// Mitsubishi GX Works2 project: PanelFlip   PLC: FX3U/FX3UC

// global labels: Global1
VAR_GLOBAL
  XXLimitN AT M8344 : BOOL;
  XXLimitP AT M8343 : BOOL;
  XXStop AT M8349 : BOOL;
  XXBusy AT M8340 : BOOL;
  XXInterruptInverse AT M8347 : BOOL;
  XXPos AT D8340 : DINT;
  XXAccelTime AT D8348 : INT;
  XXDecelTime AT D8349 : INT;
  XXLimitNView AT M0 : BOOL;
  XXLimitPView AT M1 : BOOL;
  XXPosView AT D0 : DINT;
  XXTarPos AT D2 : DINT;
  XXFeed AT D4 : DINT;
  XXTarR AT M2 : BOOL;
  XXTarRSkip AT D6 : INT;
  XXManualN AT M3 : BOOL;
  XXManualP AT M4 : BOOL;
  XXOn AT M5 : BOOL;
  XXRun AT M6 : BOOL;
  XXDirection AT M7 : BOOL;
  XXMinI AT X000 : BOOL;
  XXAlarmI AT X004 : BOOL;
  XXReadyI AT X010 : BOOL;
  XXLimitNI AT X011 : BOOL;
  XXLimitPI AT X012 : BOOL;
  XXPulseO AT Y000 : BOOL;
  XXDirectionO AT Y004 : BOOL;
  XXOnO AT Y002 : BOOL;
  MachineReady AT M8 : BOOL;
  MachineReadyTimer AT TC0 : BOOL;
  DataState AT D7 : INT;
  Run AT M9 : BOOL;
  RunStop AT M10 : BOOL;
  RunReset AT M11 : BOOL;
  RunState AT D8 : INT;
  RunStateNext AT M12 : BOOL;
  RunStateBase AT D9 : INT;
  RunStateBaseNext AT M13 : BOOL;
  RunStateGrab AT D10 : INT;
  RunStateGrabNext AT M14 : BOOL;
  RunStateFlip AT D11 : INT;
  RunStateFlipNext AT M15 : BOOL;
  FlipFoilIn AT M16 : BOOL;
  FlipFoilInI AT X001 : BOOL;
  FlipFoilInIPulseCatch AT M8171 : BOOL;
  FlipFoilInIDenoiseTimer AT TC1 : BOOL;
  FlipEnd AT M17 : BOOL;
  FlipEndI AT X002 : BOOL;
  FlipEndIPulseCatch AT M8172 : BOOL;
  RS485Index AT D12 : INT;
  RS485Timer AT TC2 : BOOL;
  RS485RW : RS485RW;
  RS485Send0 AT D13 : INT;
  RS485Send1 AT D14 : INT;
  RS485Send2 AT D15 : INT;
  RS485Send3 AT D16 : INT;
  RS485Send4 AT D17 : INT;
  RS485Send5 AT D18 : INT;
  RS485Send6 AT D19 : INT;
  RS485Send7 AT D20 : INT;
  RS485Send8 AT D21 : INT;
  RS485Send9 AT D22 : INT;
  RS485Send10 AT D23 : INT;
  RS485Send11 AT D24 : INT;
  RS485Send12 AT D25 : INT;
  RS485Send13 AT D26 : INT;
  RS485Send14 AT D27 : INT;
  RS485Send15 AT D28 : INT;
  RS485Send16 AT D29 : INT;
  RS485Send17 AT D30 : INT;
  RS485Send18 AT D31 : INT;
  RS485Send19 AT D32 : INT;
  RS485Receive0 AT D33 : INT;
  RS485Receive1 AT D34 : INT;
  RS485Receive2 AT D35 : INT;
  RS485Receive3 AT D36 : INT;
  RS485Receive4 AT D37 : INT;
  RS485Receive5 AT D38 : INT;
  RS485Receive6 AT D39 : INT;
  RS485Receive7 AT D40 : INT;
  RS485Receive8 AT D41 : INT;
  RS485Receive9 AT D42 : INT;
  RS485Receive10 AT D43 : INT;
  RS485Receive11 AT D44 : INT;
  RS485Receive12 AT D45 : INT;
  RS485Receive13 AT D46 : INT;
  RS485Receive14 AT D47 : INT;
  RS485Receive15 AT D48 : INT;
  RS485Receive16 AT D49 : INT;
  RS485Receive17 AT D50 : INT;
  RS485Receive18 AT D51 : INT;
  RS485Receive19 AT D52 : INT;
  SpindleFlipRun AT M18 : BOOL;
  SpindleFlipRunO AT Y014 : BOOL;
  SpindleBeltRun AT M19 : BOOL;
  SpindleBeltRunO AT Y015 : BOOL;
  SpindleFlip_W_HzValue0 AT D53 : INT;
  SpindleBelt_W_HzValue1 AT D54 : INT;
  SpindleFlip_W_RunValue2 AT D55 : INT;
  SpindleBelt_W_RunValue3 AT D56 : INT;
  SpindleFlip_R_HzValue4 AT D57 : INT;
  SpindleBelt_R_HzValue5 AT D58 : INT;
  SpindleFlip_R_SetHzValue6 AT D59 : INT;
  SpindleBelt_R_SetHzValue7 AT D60 : INT;
  SpindleFlip_R_BusVValue8 AT D61 : INT;
  SpindleBelt_R_BusVValue9 AT D62 : INT;
  SpindleFlip_R_OutVValue10 AT D63 : INT;
  SpindleBelt_R_OutVValue11 AT D64 : INT;
  SpindleFlip_R_OutCValue12 AT D65 : INT;
  SpindleBelt_R_OutCValue13 AT D66 : INT;
  RS485SpindleFlip_W_Hz0 AT M20 : BOOL;
  RS485SpindleBelt_W_Hz1 AT M21 : BOOL;
  RS485SpindleFlip_W_Run2 AT M22 : BOOL;
  RS485SpindleBelt_W_Run3 AT M23 : BOOL;
  RS485SpindleFlip_R_Hz4 AT M24 : BOOL;
  RS485SpindleBelt_R_Hz5 AT M25 : BOOL;
  RS485SpindleFlip_R_SetHz6 AT M26 : BOOL;
  RS485SpindleBelt_R_SetHz7 AT M27 : BOOL;
  RS485SpindleFlip_R_BusV8 AT M28 : BOOL;
  RS485SpindleBelt_R_BusV9 AT M29 : BOOL;
  RS485SpindleFlip_R_OutV10 AT M30 : BOOL;
  RS485SpindleBelt_R_OutV11 AT M31 : BOOL;
  RS485SpindleFlip_R_OutC12 AT M32 : BOOL;
  RS485SpindleBelt_R_OutC13 AT M33 : BOOL;
  RS485Dummy14 AT M34 : BOOL;
  RS485Dummy15 AT M35 : BOOL;
  GrabMoveStart AT D67 : DINT;
  GrabMoveEnd AT D69 : DINT;
  GrabMoveSpeed AT D71 : DINT;
  GrabMoveAccelTime AT D73 : INT;
  GrabMoveDecelTime AT D74 : INT;
  GrabDownMin AT M36 : BOOL;
  GrabDownMinI AT X005 : BOOL;
  GrabDownMax AT M37 : BOOL;
  GrabDownMaxI AT X006 : BOOL;
  GrabDown AT M38 : BOOL;
  GrabDownO AT Y005 : BOOL;
  GrabDownATimer AT TC3 : BOOL;
  GrabDownATimerDelay AT D75 : INT;
  GrabDownBTimer AT TC4 : BOOL;
  GrabDownBTimerDelay AT D76 : INT;
  GrabDownCTimer AT TC5 : BOOL;
  GrabDownCTimerDelay AT D77 : INT;
  GrabDownDTimer AT TC6 : BOOL;
  GrabDownDTimerDelay AT D78 : INT;
  GrabDownCXTimer AT TC7 : BOOL;
  GrabOn1 AT M39 : BOOL;
  GrabOn2 AT M40 : BOOL;
  GrabOn3 AT M41 : BOOL;
  GrabOn4 AT M42 : BOOL;
  GrabOn5 AT M43 : BOOL;
  GrabOn1O AT Y006 : BOOL;
  GrabOn2O AT Y010 : BOOL;
  GrabOn3O AT Y011 : BOOL;
  GrabOn4O AT Y012 : BOOL;
  GrabOn5O AT Y013 : BOOL;
  GrabOnTimer AT TC8 : BOOL;
  GrabOnTimerDelay AT D79 : INT;
  GrabOnIndex AT D80 : INT;
  GrabPump AT M44 : BOOL;
  GrabPumpO AT Y007 : BOOL;
  GrabManualEnable AT M45 : BOOL;
  GrabStepReady AT M46 : BOOL;
  BaseEmpty AT M47 : BOOL;
  BaseEmptyI AT X003 : BOOL;
  MirrorI AT X007 : BOOL;
  M8012PLS AT M48 : BOOL;
  TestGrabDownEnable AT M49 : BOOL;
  TestGrabDownMinTimer AT TC9 : BOOL;
  TestGrabDownMaxTimer AT TC10 : BOOL;
END_VAR

// task Task_01 (event TRUE, interval 0, priority 31): POU_01

PROGRAM POU_01
VAR
  fTmp : BOOL;
END_VAR
SET(M8002, M8336);
MOV(M8002, HFFF0, D8336);
SET(M8002, XXInterruptInverse);
ZRST(M8002, RunState, RunStateFlip);
MOV(M8002, 200, XXAccelTime);
MOV(M8002, 200, XXDecelTime);
RST(M8002, SpindleFlipRun);
RST(M8002, SpindleBeltRun);
RST(M8002, TestGrabDownEnable);

(*ready*)
RST(M8002, MachineReady);
OUT_T(NOT MachineReady, MachineReadyTimer, 10);
SET(MachineReadyTimer, MachineReady);

(*data*)
RST(M8002, DataState);
DECO(M8000, DataState, 3, M500); (*M500 - M507*)
MOV(M501, GrabMoveAccelTime, XXAccelTime);
MOV(M501, GrabMoveDecelTime, XXDecelTime);
MOV(M501, 2, DataState); (*jump to rs485 sync data*)

SET(M507 AND RunState = 0 AND Run , fTmp);
RST(fTmp, Run);
RST(fTmp, RunStop);
MOV(fTmp, 1, RunState);
RST(fTmp, fTmp);
SET(RunState > 0 AND RunReset, fTmp);
RST(fTmp, RunReset);
RST(fTmP, RunStop);
RST(fTmp, Run);
RST(fTmp, SpindleFlipRun);
RST(fTmp, SpindleBeltRun);
RST(fTmp, XXRun);
ZRST(fTmp, GrabOn1, GrabOn5);
ZRST(fTmp, RunState, RunStateFlip);
ZRST(fTmp, RunStateNext, RunStateFlipNext);
RST(fTmp, fTmp);

INC(RunStateNext, RunState);
INC(RunStateBaseNext, RunStateBase);
INC(RunStateGrabNext, RunStateGrab);
INC(RunStateFlipNext, RunStateFlip);
ZRST(M8000, RunStateNext, RunStateFlipNext);
DECO(M8000, RunState, 6, M100); 
DECO(M8000, RunStateBase, 6, M200);
DECO(M8000, RunStateGrab, 6, M300); DECO(M8000, RunStateGrab, 6, M1300); ZRST(NOT (XXTarR AND XXReadyI), M1300, M1363);
DECO(M8000, RunStateFlip, 6, M400);

(*||||||||||*)
(*||||||||||Main*)
(*start belt*)
SET(M101, SpindleBeltRun);
SET(M101, RunStateNext);
(*start belt done, start other*)
MOV(M102 AND M200, 1, RunStateBase);
MOV(M102 AND M1300, 1, RunStateGrab);
MOV(M102 AND M400, 1, RunStateFlip);
MOV(M102, 10, RunState);
(*run or stop, auto or manual*)
SET(M110 AND RunStop AND NOT BaseEmpty AND Run, fTmp);
RST(fTmp, RunStop);
RST(fTmp, Run);
RST(fTmp, fTmp);
SET(M110 AND NOT RunStop, fTmp);
MOV(fTmp AND NOT GrabManualEnable, 11, RunState);
MOV(fTmp AND GrabManualEnable, 21, RunState);
DECOP(fTmp, RunState, 6, M100);
RST(fTmp, fTmp);
(*auto*)
SET(M111 AND M1340, fTmp);
MOV(fTmp AND NOT RunStop, 11, RunStateGrab);
MOV(fTmp, 10, RunState);
SET(fTmp, GrabStepReady);
RST(fTmp, fTmp);
(*manual*)
SET(M121 AND M1340, fTmp);
MOV(fTmp AND NOT RunStop, 11, RunStateGrab);
MOV(fTmp, 10, RunState);
RST(fTmp, fTmp);
(*/////base and flip*)
(*seperate sequence*)
MOV(M219 OR M220, 11, RunStateBase);
MOV(M420, 11, RunStateFlip);

(*||||||||||*)
(*||||||||||Base*)
(*/////reset*)
MOV(M201, 11, RunStateBase);
(*empty, stop*)
MOV(M211 AND BaseEmpty, 19, RunStateBase);
SET(M211 AND BaseEmpty, RunStop);
(*not empty, ready*)
MOV(M211 AND NOT BaseEmpty, 20, RunStateBase);
(*||||||||||*)

(*||||||||||*)
(*||||||||||Grab*)
(*/////reset*)
(*1 pulse = 0.01 mm*)
(*turn servo on, grab up off all*)
SET(M301 AND NOT XXOn, XXOn);
RST(M301, GrabDown);
ZRST(M301, GrabOn1, GrabOn5);
SET(M1301 AND GrabDownMin, RunStateGrabNext);
(*min on, jump to dvit*)
MOV(M1302 AND XXMinI, 5, RunStateGrab);
(*min off, jump to move back*)
SET(M1302 AND NOT XXMinI, RunStateGrabNext);
(*move back*)
RST(M1303, XXPos);
DMOV(M1303, -3000_00, XXTarPos);
DMOV(M1303, 100_00, XXFeed);
SET(M1303, XXRun);
SET(M1303, RunStateGrabNext);
(*move back hit min, jump to dvit*)
RST(M304 AND XXMinI, XXRun);
MOV(M1304 AND XXMinI, 5, RunStateGrab);
(*dvit*)
DDVIT(M305, 10_00, 10_00, XXPulseO, XXDirection);
SET(M305 AND M8029, RunStateGrabNext);
RST(M305 AND M8029, M305);
(*get origin done, jump to (move to start position)*)
RST(M1306, XXPos);
RST(M1306, XXTarPos);
MOV(M1306, 30, RunStateGrab);
(*/////work sequence*)
(*move to start position*)
DMOV(M1311, GrabMoveStart, XXTarPos);
DMOV(M1311, GrabMoveSpeed, XXFeed);
SET(M1311, XXRun);
SET(M1311, RunStateGrabNext);
(*grab down on all, reset grab on index*)
SET(M1312, GrabDown);
SET(M1312, GrabOn1);
SET(M1312, GrabOn2);
SET(M1312, GrabOn3);
SET(M1312, GrabOn4);
SET(M1312, GrabOn5);
RST(M1312, GrabOnIndex);
SET(M1312 AND GrabDownMax, RunStateGrabNext);
(*wait A*)
OUT_T(M1313, GrabDownATimer, GrabDownATimerDelay);
SET(GrabDownATimer, RunStateGrabNext);
(*grab up*)
RST(M1314, GrabDown);
SET(M1314 AND GrabDownMin, RunStateGrabNext);
(*wait B*)
OUT_T(M1315, GrabDownBTimer, GrabDownBTimerDelay);
SET(GrabDownBTimer, RunStateGrabNext);
(*move to end position*)
DMOV(M1316, GrabMoveEnd, XXTarPos);
DMOV(M1316, GrabMoveSpeed, XXFeed);
SET(M1316, XXRun);
SET(M1316, RunStateGrabNext);
(*wait C*)
OUT_T(M1317, GrabDownCTimer, GrabDownCTimerDelay);
SET(GrabDownCTimer, RunStateGrabNext);
(*grab down*)
SET(M1318, GrabDown);
SET(M1318 AND GrabDownMax, RunStateGrabNext);
(*wait D*)
OUT_T(M1319, GrabDownDTimer, GrabDownDTimerDelay);
SET(GrabDownDTimer, RunStateGrabNext);
(*drop start*)
SET(M1320, RunStateGrabNext);
(*drop and check*)
OUT_T(M1321, GrabOnTimer, GrabOnTimerDelay);
SET(M1321 AND (GrabOnTimer OR GrabOnIndex = 0), fTmp);
RST(fTmp AND NOT MirrorI AND GrabOnIndex = 0, GrabOn1);
RST(fTmp AND NOT MirrorI AND GrabOnIndex = 1, GrabOn2);
RST(fTmp AND NOT MirrorI AND GrabOnIndex = 2, GrabOn3);
RST(fTmp AND NOT MirrorI AND GrabOnIndex = 3, GrabOn4);
RST(fTmp AND NOT MirrorI AND GrabOnIndex = 4, GrabOn5);
RST(fTmp AND MirrorI AND GrabOnIndex = 0, GrabOn5);
RST(fTmp AND MirrorI AND GrabOnIndex = 1, GrabOn4);
RST(fTmp AND MirrorI AND GrabOnIndex = 2, GrabOn3);
RST(fTmp AND MirrorI AND GrabOnIndex = 3, GrabOn2);
RST(fTmp AND MirrorI AND GrabOnIndex = 4, GrabOn1);
INC(fTmp, GrabOnIndex);
MOV(fTmp AND GrabOnIndex < 5, 20, RunStateGrab); (*jump back to (drop start)*)
MOV(fTmp AND GrabOnIndex >= 5, 22, RunStateGrab); (*drop done, use move because manual ignore RunStateGrabNext*)
RST(fTmp, fTmp);
(*grab up*)
RST(M1322, GrabDown);
SET(M1322 AND GrabDownMin, RunStateGrabNext);
(*wait C*)
OUT_T(M1323, GrabDownCXTimer, GrabDownCTimerDelay);
MOV(GrabDownCXTimer, 30, RunStateGrab);
(*move to start position*)
DMOV(M1330, GrabMoveStart, XXTarPos);
DMOV(M1330, GrabMoveSpeed, XXFeed);
SET(M1330, XXRun);
SET(M1330, RunStateGrabNext);
(*move to start position done, end*)
MOV(M1331, 40, RunStateGrab);
(*/////*)
(*manual*)
SET(GrabManualEnable AND RunStateGrabNext AND RunStateGrab > 10, fTmp);
RST(fTmp AND NOT GrabStepReady, RunStateGrabNext);
RST(fTmp AND GrabStepReady, GrabStepReady);
RST(fTmp, fTmp);
(*||||||||||*)

(*||||||||||*)
(*||||||||||Flip*)
(*/////reset*)
(*rotate, forward = 1, reverse = 2, stop = 5*)
SET(M401, SpindleFlipRun);
RST(M401, FlipEndIPulseCatch);
SET(M401, RunStateFlipNext);
(*stop rotate*)
SET(M402 AND FlipEnd, fTmp);
RST(fTmp, SpindleFlipRun);
RST(fTmp, FlipFoilInIPulseCatch);
RST(fTmp, FlipEndIPulseCatch);
MOV(fTmp, 11, RunStateFlip);
RST(fTmp, fTmp);
(*/////work sequence*)
(*foil in, rotate*)
SET(M411 AND FlipFoilIn, fTmp);
SET(fTmp, SpindleFlipRun);
RST(fTmp, FlipFoilInIPulseCatch);
RST(fTmp, FlipFoilIn);
RST(fTmp, FlipEndIPulseCatch);
SET(fTmp, RunStateFlipNext);
RST(fTmp, fTmp);
(*stop rotate*)
SET(M412 AND FlipEnd, fTmp);
RST(fTmp, SpindleFlipRun);
RST(fTmp, FlipFoilInIPulseCatch);
RST(fTmp, FlipFoilIn);
RST(fTmp, FlipEndIPulseCatch);
MOV(fTmp, 20, RunStateFlip);
RST(fTmp, fTmp);
(*||||||||||*)

(*||||||||||*)
(*||||||||||RS485*)
(*combine 2 register first 8bit data to 16bit register example: MOV(D0(High), K2M8), MOV(D1(Low), K2M0) then MOV(K4M0, D2) now D2 is combination of D0 and D1*)
(*main*)
MOV(M8002, H0C87, D8120);
MOV(M8002, K1000, D8129);
SET(M8002, M8161);
RS(M8012, RS485Send0, K8, K11, RS485Receive0);
PLS(M8012, M8012PLS); SET(M8012PLS, M8122);
RST(M8123, M8123);
(*sync data*)
DECO(M8000, RS485Index, 4, RS485SpindleFlip_W_Hz0);
(*start, set first index*)
MOV(M502, 0, RS485Index);
MOV(M502, -1, SpindleFlip_R_SetHzValue6);
MOV(M502, -1, SpindleBelt_R_SetHzValue7);
INC(M502, DataState);
(*wait, jump to set next index, exit condition*)
OUT_T(M503, RS485Timer, 5);
SET(RS485Timer AND SpindleFlip_R_SetHzValue6 = SpindleFlip_W_HzValue0 AND SpindleBelt_R_SetHzValue7 = SpindleBelt_W_HzValue1, fTmp);
MOV(RS485Timer AND fTmp, 7, DataState); (*meet condition, exit*)
INC(RS485Timer AND NOT fTmp, DataState); (*not meet condition, continue*)
RST(fTmp, fTmp);
(*set next index, back to wait*)
SET(M504 AND RS485Index = 7, fTmp);
MOV(M504 AND RS485Index = 7, 0, RS485Index);
MOV(M504 AND RS485Index = 6, 7, RS485Index);
MOV(M504 AND RS485Index = 1, 6, RS485Index);
MOV(M504 AND NOT fTmp AND RS485Index = 0, 1, RS485Index);
MOV(M504, 3, DataState);
RST(fTmp, fTmp);
(**)
(*/////spindle flip*)
RS485RW(Enable:= RS485SpindleFlip_W_Hz0, SlaveAdress:= H01, Cmd:= H06, CmdAddress:= H2001, CmdValue:= SpindleFlip_W_HzValue0, Target:= RS485Send0);
RS485RW(Enable:= RS485SpindleFlip_W_Run2, SlaveAdress:= H01, Cmd:= H06, CmdAddress:= H2000, CmdValue:= SpindleFlip_W_RunValue2, Target:= RS485Send0);
RS485RW(Enable:= RS485SpindleFlip_R_Hz4, SlaveAdress:= H01, Cmd:= H03, CmdAddress:= H3000, CmdValue:= K2, Target:= RS485Send0);
RS485RW(Enable:= RS485SpindleFlip_R_SetHz6, SlaveAdress:= H01, Cmd:= H03, CmdAddress:= H3001, CmdValue:= K2, Target:= RS485Send0);
RS485RW(Enable:= RS485SpindleFlip_R_BusV8, SlaveAdress:= H01, Cmd:= H03, CmdAddress:= H3002, CmdValue:= K2, Target:= RS485Send0);
RS485RW(Enable:= RS485SpindleFlip_R_OutV10, SlaveAdress:= H01, Cmd:= H03, CmdAddress:= H3003, CmdValue:= K2, Target:= RS485Send0);
RS485RW(Enable:= RS485SpindleFlip_R_OutC12, SlaveAdress:= H01, Cmd:= H03, CmdAddress:= H3004, CmdValue:= K2, Target:= RS485Send0);
(*/////spindle belt*)
(*spindle belt: set hz*)
RS485RW(Enable:= RS485SpindleBelt_W_Hz1, SlaveAdress:= H02, Cmd:= H06, CmdAddress:= H2001, CmdValue:= SpindleBelt_W_HzValue1, Target:= RS485Send0);
RS485RW(Enable:= RS485SpindleBelt_W_Run3, SlaveAdress:= H02, Cmd:= H06, CmdAddress:= H2000, CmdValue:= SpindleBelt_W_RunValue3, Target:= RS485Send0);
RS485RW(Enable:= RS485SpindleBelt_R_Hz5, SlaveAdress:= H02, Cmd:= H03, CmdAddress:= H3000, CmdValue:= K2, Target:= RS485Send0);
RS485RW(Enable:= RS485SpindleBelt_R_SetHz7, SlaveAdress:= H02, Cmd:= H03, CmdAddress:= H3001, CmdValue:= K2, Target:= RS485Send0);
RS485RW(Enable:= RS485SpindleBelt_R_BusV9, SlaveAdress:= H02, Cmd:= H03, CmdAddress:= H3002, CmdValue:= K2, Target:= RS485Send0);
RS485RW(Enable:= RS485SpindleBelt_R_OutV11, SlaveAdress:= H02, Cmd:= H03, CmdAddress:= H3003, CmdValue:= K2, Target:= RS485Send0);
RS485RW(Enable:= RS485SpindleBelt_R_OutC13, SlaveAdress:= H02, Cmd:= H03, CmdAddress:= H3004, CmdValue:= K2, Target:= RS485Send0);
(*move read data*)
MOV(RS485SpindleFlip_R_Hz4, RS485Receive3 * 256 + RS485Receive4, SpindleFlip_R_HzValue4);
MOV(RS485SpindleBelt_R_Hz5, RS485Receive3 * 256 + RS485Receive4, SpindleBelt_R_HzValue5);
MOV(RS485SpindleFlip_R_SetHz6, RS485Receive3 * 256 + RS485Receive4, SpindleFlip_R_SetHzValue6);
MOV(RS485SpindleBelt_R_SetHz7, RS485Receive3 * 256 + RS485Receive4, SpindleBelt_R_SetHzValue7);
MOV(RS485SpindleFlip_R_BusV8, RS485Receive3 * 256 + RS485Receive4, SpindleFlip_R_BusVValue8);
MOV(RS485SpindleBelt_R_BusV9, RS485Receive3 * 256 + RS485Receive4, SpindleBelt_R_BusVValue9);
MOV(RS485SpindleFlip_R_OutV10, RS485Receive3 * 256 + RS485Receive4, SpindleFlip_R_OutVValue10);
MOV(RS485SpindleBelt_R_OutV11, RS485Receive3 * 256 + RS485Receive4, SpindleBelt_R_OutVValue11);
MOV(RS485SpindleFlip_R_OutC12, RS485Receive3 * 256 + RS485Receive4, SpindleFlip_R_OutCValue12);
MOV(RS485SpindleBelt_R_OutC13, RS485Receive3 * 256 + RS485Receive4, SpindleBelt_R_OutCValue13);
(**)

(*||||||||||*)
RST(XXRun AND XXTarPos = XXPos, XXRun);
DDRVA(XXRun, XXTarPos, XXFeed, XXPulseO, XXDirection);
RST(M8029, XXRun);
OUT((MirrorI OR XXDirection) <> (MirrorI AND XXDirection), XXDirectionO);
INC(NOT XXRun AND NOT XXBusy AND XXTarRSkip < 5, XXTarRSkip);
RST(XXRun, XXTarRSkip);
OUT(XXTarRSkip >= 5, XXTarR);
SET(NOT MirrorI AND NOT XXLimitNI, XXLimitN); RST(NOT MirrorI AND XXLimitNI, XXLimitN);
SET(NOT MirrorI AND NOT XXLimitPI, XXLimitP); RST(NOT MirrorI AND XXLimitPI, XXLimitP);
SET(MirrorI AND NOT XXLimitNI, XXLimitP); RST(MirrorI AND XXLimitNI, XXLimitP);
SET(MirrorI AND NOT XXLimitPI, XXLimitN); RST(MirrorI AND XXLimitPI, XXLimitN);
RST(XXLimitN OR XXLimitP, XXRun);
(*||||||||||*)
DMOV(M8012, XXPos, XXPosView);
OUT(XXLimitN, XXLimitNView);
OUT(XXLimitP, XXLimitPView);

(*Input*)
OUT(BaseEmptyI, BaseEmpty);
SET(NOT TestGrabDownEnable AND GrabDownMinI, GrabDownMin); RST(NOT TestGrabDownEnable AND GrabDownMinI, GrabDownMax);
SET(NOT TestGrabDownEnable AND GrabDownMaxI, GrabDownMax); RST(NOT TestGrabDownEnable AND GrabDownMaxI, GrabDownMin);
OUT_T(TestGrabDownEnable AND NOT GrabDown, TestGrabDownMinTimer, 5); SET(TestGrabDownMinTimer, GrabDownMin); RST(TestGrabDownMinTimer, GrabDownMax);
OUT_T(TestGrabDownEnable AND GrabDown, TestGrabDownMaxTimer, 5); SET(TestGrabDownMaxTimer, GrabDownMax); RST(TestGrabDownMaxTimer, GrabDownMin);

EI(TRUE);
(*OUT(FlipFoilInIPulseCatch, FlipFoilIn);*)
OUT(FlipEndIPulseCatch, FlipEnd);
DI(TRUE);
OUT_T(FlipFoilInI, FlipFoilInIDenoiseTimer, 1);
SET(NOT FlipFoilIn AND FlipFoilInIDenoiseTimer, FlipFoilIn);

(*Output*)
OUT(XXOn, XXOnO);
OUT(SpindleFlipRun, SpindleFlipRunO);
OUT(SpindleBeltRun, SpindleBeltRunO);
OUT(GrabPump, GrabPumpO);
OUT(GrabDown, GrabDownO);
OUT(GrabOn1, GrabOn1O);
OUT(GrabOn2, GrabOn2O);
OUT(GrabOn3, GrabOn3O);
OUT(GrabOn4, GrabOn4O);
OUT(GrabOn5, GrabOn5O);
END_PROGRAM

FUNCTION_BLOCK RS485RW
VAR_INPUT
  SlaveAdress : INT;
  Cmd : INT;
  CmdAddress : INT;
  CmdValue : INT;
END_VAR
VAR_OUTPUT
  Target : INT;
END_VAR
VAR_INPUT
  Enable : BOOL;
END_VAR
VAR
  Buffer : ARRAY [0..7] OF INT;
END_VAR
MOV(Enable, SlaveAdress, Buffer[0]);
MOV(Enable, Cmd, Buffer[1]);
MOV(Enable, CmdAddress / 256, Buffer[2]);
MOV(Enable, CmdAddress MOD 256, Buffer[3]);
MOV(Enable, CmdValue / 256, Buffer[4]);
MOV(Enable, CmdValue MOD 256, Buffer[5]);
CRC(Enable, Buffer[0], K6, Buffer[6]);
BMOV(Enable, Buffer[0], K8, Target);
END_FUNCTION_BLOCK
